Staubli VAL3: remGetMode.pgx

program remGetMode(string& sReturn[] (dimensions=1))
  local string sMode
begin
  // Return the movement mode for remote moves
  //
  logMsg("call remGetMode")
  if bMoveLinear
    sMode="LINEAR"
  else
    sMode="OPTIMAL"
  endIf
  sReturn="GETMODE "+sMode
end
